KUKA KRL program: find_seam.src, find_seam.dat

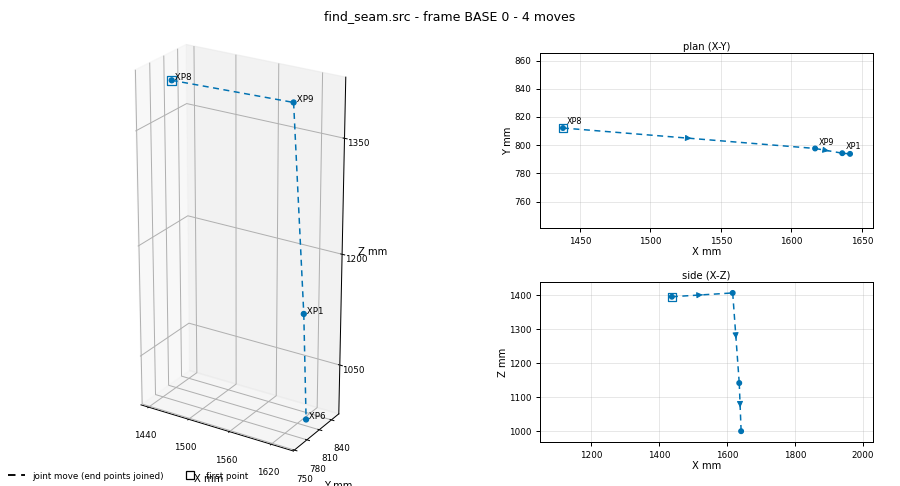
[picture p0: tool path of find_seam.src in frame BASE 0, 4 of 5 moves have a stored position in this frame; points joined in program order, loops and branches not executed]
--- find_seam.src ---
&ACCESS RVO1
&REL 1
&PARAM DISKPATH = KRC:\R1\Program\Production
DEF find_seam( )
   ;FOLD INI;%{PE}
      ;FOLD BASISTECH INI
         GLOBAL INTERRUPT DECL 3 WHEN $STOPMESS==TRUE DO IR_STOPM ( )
         INTERRUPT ON 3
         BAS (#INITMOV,0 )
      ;ENDFOLD (BASISTECH INI)
      ;FOLD USER INI
         ;Make your modifications here

      ;ENDFOLD (USER INI)
   ;ENDFOLD (INI)

   Xdummy_point = $POS_ACT
   PTP Xdummy_point

   actualHeightOffset = 10.0

   IF (NOT $IN_HOME) THEN
      HomePos()
   ENDIF

;FOLD SPTP P8 Vel=30 % PDAT9 Tool[1]:laser Base[0];%{PE}%R 8.3.38,%MKUKATPBASIS,%CSPLINE,%VSPTP_SB,%P 1:SPTP_SB, 2:P8, 3:, 5:30, 7:PDAT9
SPTP XP8 WITH $VEL_AXIS[1]= SVEL_JOINT( 30), $TOOL= STOOL2( FP8), $BASE= SBASE( FP8.BASE_NO),$IPO_MODE= SIPO_MODE( FP8.IPO_FRAME), $LOAD= SLOAD( FP8.TOOL_NO), $ACC_AXIS[1]= SACC_JOINT( PPDAT9), $GEAR_JERK[1]= SGEAR_JERK( PPDAT9)
;ENDFOLD

   ;FOLD HandShake[21 : At Hold Pos 1], WAIT on Response
      HandShake_Set (21,false)
      HandShake_Check (21,false)
   ;ENDFOLD

   nType = Task_Selection(0)

   SWITCH nType

      CASE 2

;FOLD SPTP P9 Vel=30 % PDAT10 Tool[1]:laser Base[0];%{PE}%R 8.3.38,%MKUKATPBASIS,%CSPLINE,%VSPTP_SB,%P 1:SPTP_SB, 2:P9, 3:, 5:30, 7:PDAT10
SPTP XP9 WITH $VEL_AXIS[1]= SVEL_JOINT( 30), $TOOL= STOOL2( FP9), $BASE= SBASE( FP9.BASE_NO),$IPO_MODE= SIPO_MODE( FP9.IPO_FRAME), $LOAD= SLOAD( FP9.TOOL_NO), $ACC_AXIS[1]= SACC_JOINT( PPDAT10), $GEAR_JERK[1]= SGEAR_JERK( PPDAT10)
;ENDFOLD
         fixedUpDownMove = barrel72ich
      CASE 3

;FOLD PTP P1 Vel=30 % PDAT2 Tool[1]:laser Base[0];%{PE}%R 8.3.38,%MKUKATPBASIS,%CMOVE,%VPTP,%P 1:PTP, 2:P1, 3:, 5:30, 7:PDAT2
$BWDSTART=FALSE
PDAT_ACT=PPDAT2
FDAT_ACT=FP1
BAS(#PTP_PARAMS,30)
PTP XP1
;ENDFOLD

         fixedUpDownMove = barrel60inch

      CASE 4
;FOLD PTP P6 Vel=30 % PDAT7 Tool[1]:laser Base[0];%{PE}%R 8.3.38,%MKUKATPBASIS,%CMOVE,%VPTP,%P 1:PTP, 2:P6, 3:, 5:30, 7:PDAT7
$BWDSTART=FALSE
PDAT_ACT=PPDAT7
FDAT_ACT=FP6
BAS(#PTP_PARAMS,30)
PTP XP6
;ENDFOLD
        fixedUpDownMove = barrel54inch

      DEFAULT
         RETURN

   ENDSWITCH


   LASER_APPROACH(FALSE)
   ;FOLD HandShake[22 : Barrel Found], WAIT on Response
      HandShake_Set (22,false)
      HandShake_Check (22,false)
   ;ENDFOLD

   ;Get close to the seam

   IF seamTrackDisabled <> TRUE THEN
      LASER_APPROACH(TRUE)
   ENDIF


   ;FOLD HandShake[23 : AT the Seam adjust changes], WAIT on Response
      HandShake_Set (23,false)
      HandShake_Check (23,false)
   ;ENDFOLD

   ;SEAM FOUND

   Exit_Program()

END

--- find_seam.dat ---
&ACCESS RVO1
&REL 1
&PARAM DISKPATH = KRC:\R1\Program\Production
DEFDAT  find_seam
;FOLD EXTERNAL DECLARATIONS;%{PE}%MKUKATPBASIS,%CEXT,%VCOMMON,%P
;FOLD BASISTECH EXT;%{PE}%MKUKATPBASIS,%CEXT,%VEXT,%P
EXT  BAS (BAS_COMMAND  :IN,REAL  :IN )
;ENDFOLD (BASISTECH EXT)
;FOLD USER EXT;%{E}%MKUKATPUSER,%CEXT,%VEXT,%P
;Make your modifications here
;ENDFOLD (USER EXT)
;ENDFOLD (EXTERNAL DECLARATIONS)

DECL BOOL throwawaybool
DECL REAL barrel54inch=18.0000
DECL REAL barrel60inch=12.0000
DECL REAL barrel72ich=0.0
DECL REAL fixedUpDownMove=0.0

DECL INT nType

DECL FDAT FHOME2={TOOL_NO 1,BASE_NO 0,IPO_FRAME #BASE,POINT2[] " "}
DECL PDAT PPDAT1={VEL 1.00000,ACC 5.00000,APO_DIST 100.000,APO_MODE #CDIS,GEAR_JERK 50.0000,EXAX_IGN 0}

DECL E6POS XP1={X 1636.14819,Y 794.290955,Z 1142.45789,A -6.91767406,B -89.6694489,C -178.248367,S 2,T 43,E1 0.0,E2 0.0,E3 0.0,E4 0.0,E5 0.0,E6 0.0}
DECL BASIS_SUGG_T LAST_BASIS={POINT1[] "P9                      ",POINT2[] "P9                      ",CP_PARAMS[] "CPDAT0                  ",PTP_PARAMS[] "PDAT10                  ",CONT[] "                        ",CP_VEL[] "2.0                     ",PTP_VEL[] "30                      ",SYNC_PARAMS[] "SYNCDAT                 ",SPL_NAME[] "S0                      ",A_PARAMS[] "ADAT0                   "}
DECL FDAT FP1={TOOL_NO 1,BASE_NO 0,IPO_FRAME #BASE,POINT2[] " ",TQ_STATE FALSE}
DECL PDAT PPDAT2={VEL 100.000,ACC 5.00000,APO_DIST 100.000,APO_MODE #CDIS,GEAR_JERK 50.0000,EXAX_IGN 0}
DECL E6POS XP2={X 511.514648,Y 1400.11133,Z 1349.18750,A -164.725632,B -89.6085205,C 114.340492,S 6,T 51,E1 0.0,E2 0.0,E3 0.0,E4 0.0,E5 0.0,E6 0.0}
DECL FDAT FP2={TOOL_NO 1,BASE_NO 0,IPO_FRAME #BASE,POINT2[] " ",TQ_STATE FALSE}
DECL PDAT PPDAT3={VEL 100.000,ACC 5.00000,APO_DIST 100.000,APO_MODE #CDIS,GEAR_JERK 50.0000,EXAX_IGN 0}
DECL E6POS XP3={X 522.845825,Y 1446.49805,Z 1770.12634,A 128.793320,B 0.164586022,C -179.744675,S 18,T 43,E1 0.0,E2 0.0,E3 0.0,E4 0.0,E5 0.0,E6 0.0}
DECL FDAT FP3={TOOL_NO 1,BASE_NO 0,IPO_FRAME #BASE,POINT2[] " ",TQ_STATE FALSE}
DECL PDAT PPDAT4={VEL 100.000,ACC 5.00000,APO_DIST 100.000,APO_MODE #CDIS,GEAR_JERK 50.0000,EXAX_IGN 0}
DECL E6POS XP4={X 522.711853,Y 1445.53809,Z 1575.23364,A 128.791397,B 0.166948795,C -179.743484,S 18,T 43,E1 0.0,E2 0.0,E3 0.0,E4 0.0,E5 0.0,E6 0.0}
DECL FDAT FP4={TOOL_NO 1,BASE_NO 0,IPO_FRAME #BASE,POINT2[] " ",TQ_STATE FALSE}
DECL PDAT PPDAT5={VEL 100.000,ACC 100.000,APO_DIST 100.000,APO_MODE #CDIS,GEAR_JERK 50.0000,EXAX_IGN 0}
DECL E6POS XP5={X 518.601135,Y 1451.07666,Z 1600.39282,A 128.791641,B 0.166907653,C -179.742844,S 18,T 43,E1 0.0,E2 0.0,E3 0.0,E4 0.0,E5 0.0,E6 0.0}
DECL FDAT FP5={TOOL_NO 1,BASE_NO 0,IPO_FRAME #BASE,POINT2[] " ",TQ_STATE FALSE}
DECL PDAT PPDAT6={VEL 100.000,ACC 100.000,APO_DIST 100.000,APO_MODE #CDIS,GEAR_JERK 50.0000,EXAX_IGN 0}
DECL E6POS XP6={X 1641.65686,Y 793.818,Z 1000.77246,A -6.91767263,B -89.6694489,C -178.248383,S 2,T 43,E1 0.0,E2 0.0,E3 0.0,E4 0.0,E5 0.0,E6 0.0}
DECL FDAT FP6={TOOL_NO 1,BASE_NO 0,IPO_FRAME #BASE,POINT2[] " ",TQ_STATE FALSE}
DECL PDAT PPDAT7={VEL 100.000,ACC 5.00000,APO_DIST 100.000,APO_MODE #CDIS,GEAR_JERK 50.0000,EXAX_IGN 0}
DECL E6POS XP7={X 1088.80115,Y 847.245361,Z 1230.66431,A -164.726181,B -89.6085205,C 110.339455,S 6,T 51,E1 0.0,E2 0.0,E3 0.0,E4 0.0,E5 0.0,E6 0.0}
DECL FDAT FP7={TOOL_NO 1,BASE_NO 0,IPO_FRAME #BASE,POINT2[] " ",TQ_STATE FALSE}
DECL PDAT PPDAT8={VEL 100.000,ACC 5.00000,APO_DIST 100.000,APO_MODE #CDIS,GEAR_JERK 50.0000,EXAX_IGN 0}
DECL E6POS XP8={X 1438.03943,Y 812.157104,Z 1396.17175,A -6.91768074,B -89.6694489,C -178.248367,S 2,T 43,E1 0.0,E2 0.0,E3 0.0,E4 0.0,E5 0.0,E6 0.0}
DECL FDAT FP8={TOOL_NO 1,BASE_NO 0,IPO_FRAME #BASE,POINT2[] " ",TQ_STATE FALSE}
DECL PDAT PPDAT9={VEL 100.000,ACC 5.00000,APO_DIST 100.000,APO_MODE #CDIS,GEAR_JERK 50.0000,EXAX_IGN 0}
DECL E6POS XP9={X 1616.87598,Y 797.652161,Z 1407.33948,A -13.7988110,B -89.8405304,C -168.316452,S 2,T 43,E1 0.0,E2 0.0,E3 0.0,E4 0.0,E5 0.0,E6 0.0}
DECL FDAT FP9={TOOL_NO 1,BASE_NO 0,IPO_FRAME #BASE,POINT2[] " ",TQ_STATE FALSE}
DECL PDAT PPDAT10={VEL 100.000,ACC 5.00000,APO_DIST 100.000,APO_MODE #CDIS,GEAR_JERK 50.0000,EXAX_IGN 0}
ENDDAT
